{attribute 'qualified_only'}
{attribute 'strict'}
TYPE CircuitBreakerStatus :
(
	OFF        := 0, // Channel has been set OFF either manually or programatically (only available in bidirectional mode)
	ON         := 1, // Channel is ON and funcioning normally (only available in bidirectional mode)
	TRIPPED    := 2, // An overcurrent event has tripped the device
	RESET      := 3, // A reset signal has been sent to the device but it hasn't responded yet
	UNKNOWN    := 4, // Comms isssue, data not yet recived, 
	NOTTRIPPED := 5  // Channel is OFF or ON (only available in unidirectional mode)  
);
END_TYPE

(* stored: Version 1.1.0.1, ProductVersion 3.1.4024.15
   EnumerationTextList CircuitBreakerStatus: Id {1ff68e56-cae4-41db-870f-2360cfc5ceed} *)
